FUNCTION_BLOCK CALC_ITERATIONS
  (* Standard: 61499-2 *)
  (* Version 1.0, 31/05/2012, GASR *)
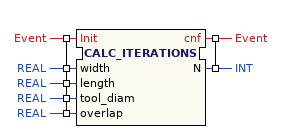
  EVENT_INPUT
    Init WITH width, length, tool_diam, overlap;
  END_EVENT
  EVENT_OUTPUT
    cnf WITH N;
  END_EVENT
  VAR_INPUT
    width : REAL;
    length : REAL;
    tool_diam : REAL;
    overlap : REAL;
  END_VAR
  VAR_OUTPUT
    N : INT;
  END_VAR
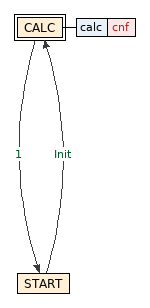
  EC_STATES
    CALC : calc -> cnf;
    START;
  END_STATES
  EC_TRANSITIONS
    CALC TO START := 1;
    START TO CALC := Init;
  END_TRANSITIONS
  ALGORITHM calc IN Lua:
				if not tonumber(overlap) then
					overlap = 0
				end
				local a = width
				if length > width then
					a = length
				end
				N = (0.5*a - tool_diam)/(tool_diam - overlap)
				N = ceil(N)
  END_ALGORITHM
END_FUNCTION_BLOCK
